// TIA Portal project "Sort By Shape & Color" (V16)
// Vorlageprojekt für das Buch mit Zielsystem S7-1200

(* hardware
DEVICE "S7-1200-Station_1"  S7-1200 Station
   slot 0: "Baugruppenträger_0"  Rack  V1.0
   slot 1: "PLC_1"  CPU 1211C DC/DC/DC  6ES7 211-1AE40-0XB0  V4.1
*)

// ===== PLC "PLC_1"  CPU 1211C DC/DC/DC =====

VAR_GLOBAL   // PLC tag table "Standard-Variablentabelle"
   "belt 6m 1" AT %A0.0 : Bool;
   "start" AT %E0.0 : Bool;
   "stop" AT %E0.1 : Bool;
   "Tag_4" AT %I10.0 : Bool;
   "Tag_5" AT %Q10.0 : Bool;
   "Tag_6" AT %I10.1 : Bool;
   "X" AT %M0.0 : Bool;
   "belt 2m 1" AT %Q0.1 : Bool;
   "belt 2m 2" AT %Q0.2 : Bool;
   "vision1" AT %I0.2 : Bool;
   "pivot1" AT %Q0.6 : Bool;
   "pivot1 +" AT %Q0.7 : Bool;
   "vision3" AT %I0.4 : Bool;
   "vision2" AT %I0.3 : Bool;
   "Tag_1" AT %M0.2 : Bool;
   "Y" AT %M0.1 : Bool;
   "timer2 marker" AT %M0.3 : Bool;
   "pivot2" AT %Q1.0 : Bool;
   "pivot2 +" AT %Q1.1 : Bool;
   "t1 marker" AT %M0.4 : Bool;
   "ccw" AT %Q0.5 : Bool;
   "belt 2m 3" AT %Q0.3 : Bool;
   "belt 2m 4" AT %Q0.4 : Bool;
   "pivot3 +" AT %Q1.3 : Bool;
   "vision4" AT %I0.5 : Bool;
   "pivot3" AT %Q1.2 : Bool;
   "Tag_2" AT %M0.5 : Bool;
   "Start Light" AT %Q1.4 : Bool;
   "Stop Light" AT %Q1.5 : Bool;
END_VAR

// folder: System blocks/Program resources

DATA_BLOCK "T2"   // DB1
{ S7_Optimized_Access := 'TRUE' }
AUTHOR : Simatic
FAMILY : IEC
NAME : IEC_TMR
VERSION : 1.0
// stored: InstanceOfName IEC_TIMER
"IEC_TIMER"
BEGIN
END_DATA_BLOCK

DATA_BLOCK "T1"   // DB2
{ S7_Optimized_Access := 'TRUE' }
AUTHOR : Simatic
FAMILY : IEC
NAME : IEC_TMR
VERSION : 1.0
// stored: InstanceOfName IEC_TIMER
"IEC_TIMER"
BEGIN
END_DATA_BLOCK

DATA_BLOCK "T3"   // DB3
{ S7_Optimized_Access := 'TRUE' }
AUTHOR : Simatic
FAMILY : IEC
NAME : IEC_TMR
VERSION : 1.0
// stored: InstanceOfName IEC_TIMER
"IEC_TIMER"
BEGIN
END_DATA_BLOCK

// folder: (top level)

FUNCTION "MHJ-PLC-Lab-Function-S71200" : Void   // FC9000, SCL
{ S7_Optimized_Access := 'TRUE' }
VERSION : 0.1
   VAR_TEMP
      rdTimeReturn : Int;
      outputTime : DTL;
      SyncVal : Byte;
      forVal : Int;
      forVal_2 : Int;
      Value : Byte;
   END_VAR
   VAR CONSTANT
      CompVal : Byte := 16#34;
      Value_01 : Byte := 16#11;
      Value_01_DW : DWord := 16#A165_D992;
      Value_02_DW : DWord := 16#58BE_4401;
   END_VAR
BEGIN

   #Value:=PEEK(area := 16#82,
        dbNumber := 0,
        byteOffset := 511);
   #Value := #Value + 1;

   POKE(area := 16#82,
        dbNumber := 0,
        byteOffset := 511,
        value := #Value);

   POKE(area:=16#81,
        dbNumber:=0,
        byteOffset:=1016,
        value:=#Value_01_DW);
   POKE(area := 16#81,
        dbNumber := 0,
        byteOffset := 1020,
        value := #Value_02_DW);

   POKE(area := 16#81,
        dbNumber := 0,
        byteOffset := 511,
        value := B#16#00);

   FOR #forVal := 0 TO 120 DO
       FOR #forVal_2:=0 TO 10 DO
           #rdTimeReturn:=RD_SYS_T(#outputTime);
           #rdTimeReturn := WR_SYS_T(#outputTime);
           #rdTimeReturn := RD_SYS_T(#outputTime);
           #rdTimeReturn := WR_SYS_T(#outputTime);
       END_FOR;
       #SyncVal:= PEEK(area := 16#81,
                      dbNumber := 0,
                      byteOffset := 511);
       IF #SyncVal = #CompVal THEN
          GOTO M_1;
       END_IF;
   END_FOR;
   RETURN;

   M_1:
   POKE(area := 16#81,
        dbNumber := 0,
        byteOffset := 511,
        value := B#16#0);
END_FUNCTION

ORGANIZATION_BLOCK "Main"   // OB1, LAD, ProgramCycle
TITLE = "Main Program Sweep (Cycle)"
{ S7_Optimized_Access := 'TRUE' }
VERSION : 0.1
   VAR_INPUT
      Initial_Call : Bool;   // Initial call of this OB
      Remanence : Bool;   // =True, if remanent data are available
   END_VAR
BEGIN

REGION Network 1: Konnektierungsbaustein für PLC-Lab
   // Im Netzwerk 1 wird der Konnektierungsbaustein für PLC-Lab aufgerufen.
   // Dieser Aufruf darf nicht entfernt werden!
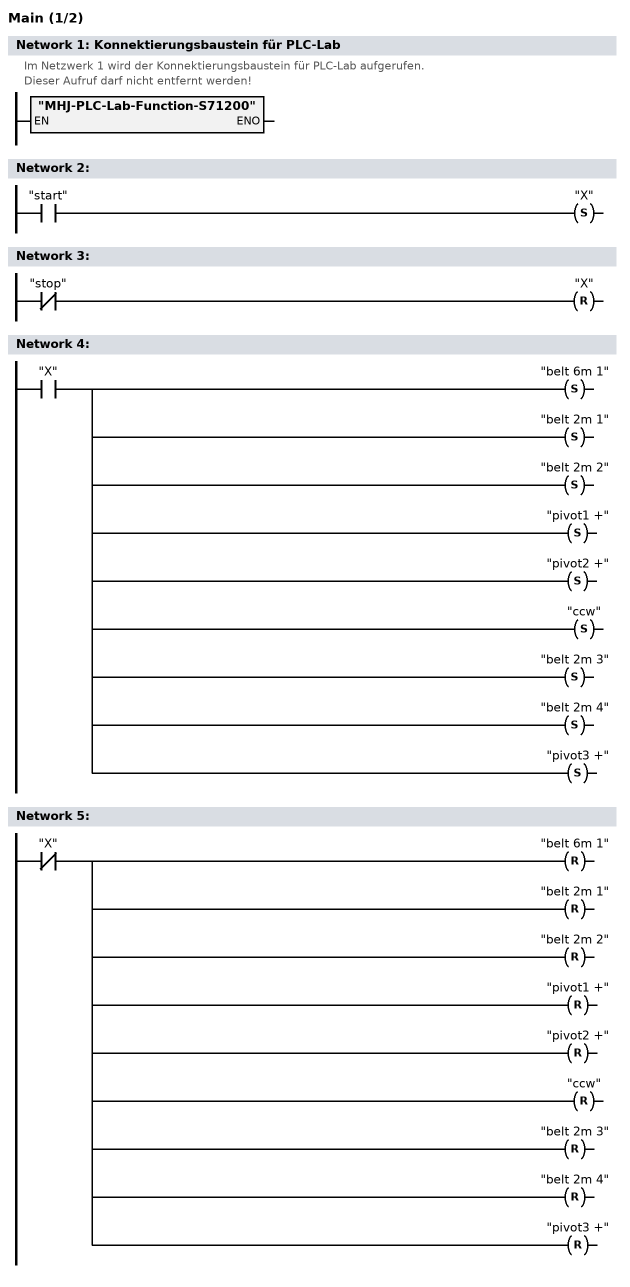
   RUNG wire#powerrail
      "MHJ-PLC-Lab-Function-S71200"()
   END_RUNG
   // the same network as SCL:
   "MHJ-PLC-Lab-Function-S71200"();
END_REGION

REGION Network 2
   RUNG wire#powerrail
      Contact( "start" )
      S_Coil( "X" )
   END_RUNG
   // the same network as SCL:
   IF "start" THEN "X" := TRUE; END_IF;
END_REGION

REGION Network 3
   RUNG wire#powerrail
      I_Contact( "stop" )
      R_Coil( "X" )
   END_RUNG
   // the same network as SCL:
   IF NOT "stop" THEN "X" := FALSE; END_IF;
END_REGION

REGION Network 4
   RUNG wire#powerrail
      Contact( "X" )
      wire#w1
      S_Coil( "belt 6m 1" )
   END_RUNG
   RUNG wire#w1
      S_Coil( "belt 2m 1" )
   END_RUNG
   RUNG wire#w1
      S_Coil( "belt 2m 2" )
   END_RUNG
   RUNG wire#w1
      S_Coil( "pivot1 +" )
   END_RUNG
   RUNG wire#w1
      S_Coil( "pivot2 +" )
   END_RUNG
   RUNG wire#w1
      S_Coil( "ccw" )
   END_RUNG
   RUNG wire#w1
      S_Coil( "belt 2m 3" )
   END_RUNG
   RUNG wire#w1
      S_Coil( "belt 2m 4" )
   END_RUNG
   RUNG wire#w1
      S_Coil( "pivot3 +" )
   END_RUNG
   // the same network as SCL:
   IF "X" THEN
       "belt 6m 1" := TRUE;
       "belt 2m 1" := TRUE;
       "belt 2m 2" := TRUE;
       "pivot1 +" := TRUE;
       "pivot2 +" := TRUE;
       "ccw" := TRUE;
       "belt 2m 3" := TRUE;
       "belt 2m 4" := TRUE;
       "pivot3 +" := TRUE;
   END_IF;
END_REGION

REGION Network 5
   RUNG wire#powerrail
      I_Contact( "X" )
      wire#w1
      R_Coil( "belt 6m 1" )
   END_RUNG
   RUNG wire#w1
      R_Coil( "belt 2m 1" )
   END_RUNG
   RUNG wire#w1
      R_Coil( "belt 2m 2" )
   END_RUNG
   RUNG wire#w1
      R_Coil( "pivot1 +" )
   END_RUNG
   RUNG wire#w1
      R_Coil( "pivot2 +" )
   END_RUNG
   RUNG wire#w1
      R_Coil( "ccw" )
   END_RUNG
   RUNG wire#w1
      R_Coil( "belt 2m 3" )
   END_RUNG
   RUNG wire#w1
      R_Coil( "belt 2m 4" )
   END_RUNG
   RUNG wire#w1
      R_Coil( "pivot3 +" )
   END_RUNG
   // the same network as SCL:
   IF NOT "X" THEN
       "belt 6m 1" := FALSE;
       "belt 2m 1" := FALSE;
       "belt 2m 2" := FALSE;
       "pivot1 +" := FALSE;
       "pivot2 +" := FALSE;
       "ccw" := FALSE;
       "belt 2m 3" := FALSE;
       "belt 2m 4" := FALSE;
       "pivot3 +" := FALSE;
   END_IF;
END_REGION

REGION Network 6
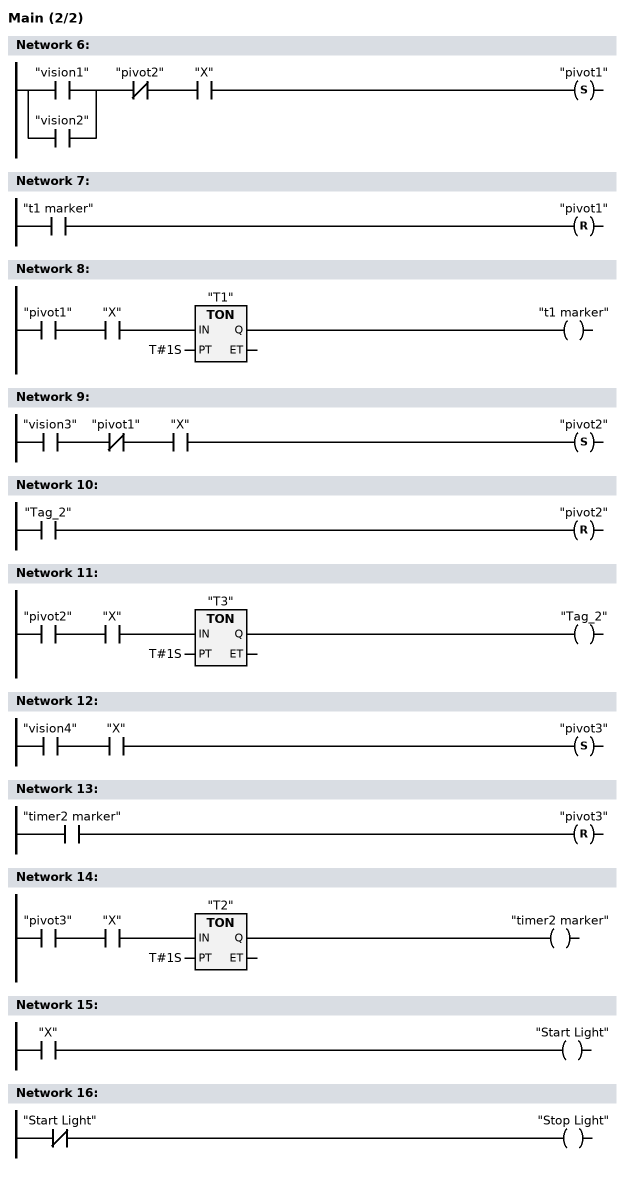
   RUNG wire#powerrail
      Contact( "vision1" )
      wire#w1
      I_Contact( "pivot2" )
      Contact( "X" )
      S_Coil( "pivot1" )
   END_RUNG
   RUNG wire#powerrail
      Contact( "vision2" )
   END_RUNG wire#w1
   // the same network as SCL:
   IF ("vision1" OR "vision2") AND NOT "pivot2" AND "X" THEN "pivot1" := TRUE; END_IF;
END_REGION

REGION Network 7
   RUNG wire#powerrail
      Contact( "t1 marker" )
      R_Coil( "pivot1" )
   END_RUNG
   // the same network as SCL:
   IF "t1 marker" THEN "pivot1" := FALSE; END_IF;
END_REGION

REGION Network 8
   "T1".TON(IN := "pivot1" AND "X", PT := T#1S);
   "t1 marker" := "T1".Q;
END_REGION

REGION Network 9
   RUNG wire#powerrail
      Contact( "vision3" )
      I_Contact( "pivot1" )
      Contact( "X" )
      S_Coil( "pivot2" )
   END_RUNG
   // the same network as SCL:
   IF "vision3" AND NOT "pivot1" AND "X" THEN "pivot2" := TRUE; END_IF;
END_REGION

REGION Network 10
   RUNG wire#powerrail
      Contact( "Tag_2" )
      R_Coil( "pivot2" )
   END_RUNG
   // the same network as SCL:
   IF "Tag_2" THEN "pivot2" := FALSE; END_IF;
END_REGION

REGION Network 11
   "T3".TON(IN := "pivot2" AND "X", PT := T#1S);
   "Tag_2" := "T3".Q;
END_REGION

REGION Network 12
   RUNG wire#powerrail
      Contact( "vision4" )
      Contact( "X" )
      S_Coil( "pivot3" )
   END_RUNG
   // the same network as SCL:
   IF "vision4" AND "X" THEN "pivot3" := TRUE; END_IF;
END_REGION

REGION Network 13
   RUNG wire#powerrail
      Contact( "timer2 marker" )
      R_Coil( "pivot3" )
   END_RUNG
   // the same network as SCL:
   IF "timer2 marker" THEN "pivot3" := FALSE; END_IF;
END_REGION

REGION Network 14
   "T2".TON(IN := "pivot3" AND "X", PT := T#1S);
   "timer2 marker" := "T2".Q;
END_REGION

REGION Network 15
   RUNG wire#powerrail
      Contact( "X" )
      Coil( "Start Light" )
   END_RUNG
   // the same network as SCL:
   "Start Light" := "X";
END_REGION

REGION Network 16
   RUNG wire#powerrail
      I_Contact( "Start Light" )
      Coil( "Stop Light" )
   END_RUNG
   // the same network as SCL:
   "Stop Light" := NOT "Start Light";
END_REGION
END_ORGANIZATION_BLOCK